// Mitsubishi GX Works2 project: code_project_big   PLC: FX3U/FX3UC

PROGRAM MAIN
VAR
  auto : BOOL;
END_VAR
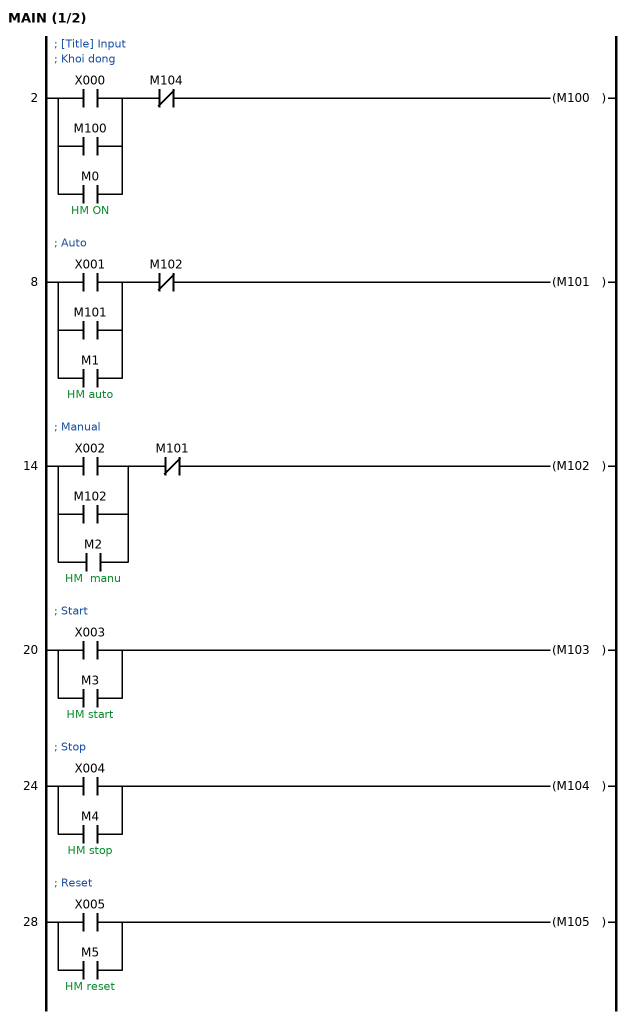
; [Title] Input
; Khoi dong
2     LD      X000
      OR      M100
      OR      M0  ; HM ON
      ANI     M104
      OUT     M100
; Auto
8     LD      X001
      OR      M101
      OR      M1  ; HM auto
      ANI     M102
      OUT     M101
; Manual
14    LD      X002
      OR      M102
      OR      M2  ; HM  manu
      ANI     M101
      OUT     M102
; Start
20    LD      X003
      OR      M3  ; HM start
      OUT     M103
; Stop
24    LD      X004
      OR      M4  ; HM stop
      OUT     M104
; Reset
28    LD      X005
      OR      M5  ; HM reset
      OUT     M105
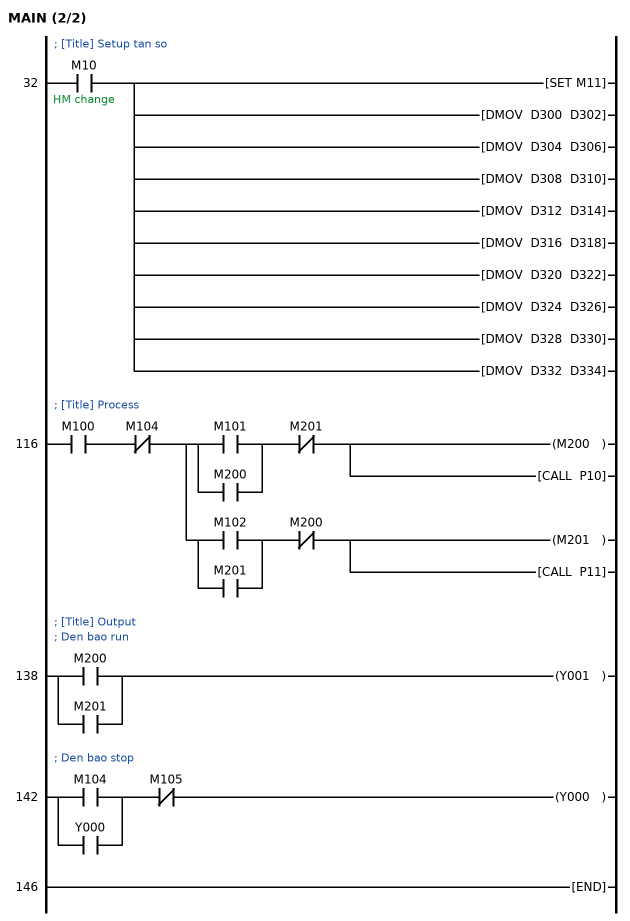
; [Title] Setup tan so
32    LD      M10  ; HM change
      SET     M11
      DMOV    D300 D302
      DMOV    D304 D306
      DMOV    D308 D310
      DMOV    D312 D314
      DMOV    D316 D318
      DMOV    D320 D322
      DMOV    D324 D326
      DMOV    D328 D330
      DMOV    D332 D334
; [Title] Process
116   LD      M100
      ANI     M104
      MPS
      LD      M101
      OR      M200
      ANB
      ANI     M201
      OUT     M200
      CALL    P10
      MPP
      LD      M102
      OR      M201
      ANB
      ANI     M200
      OUT     M201
      CALL    P11
; [Title] Output
; Den bao run
138   LD      M200
      OR      M201
      OUT     Y001
; Den bao stop
142   LD      M104
      OR      Y000
      ANI     M105
      OUT     Y000
146   END
END_PROGRAM

PROGRAM auto
VAR
  auto : POINTER;  (* ctr con *)
END_VAR
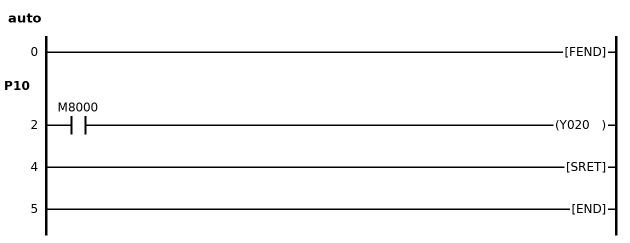
0     FEND
      P10
2     LD      M8000
      OUT     Y020
4     SRET
5     END
END_PROGRAM

PROGRAM manual
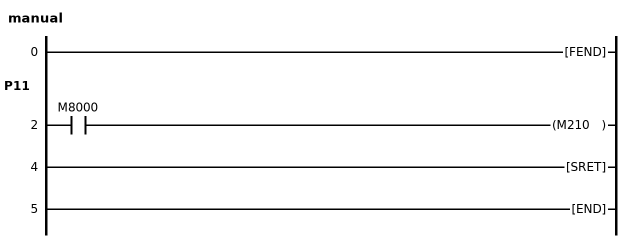
0     FEND
      P11
2     LD      M8000
      OUT     M210
4     SRET
5     END
END_PROGRAM
